# EPICS autosave request: iocBoot/iocCARSPil3Table/auto_settings.req
file "CARS_motor_settings.req",       P=$(P), M=m1
file "CARS_motor_settings.req",       P=$(P), M=m2
file "CARS_motor_settings.req",       P=$(P), M=m3
file "CARS_motor_settings.req",       P=$(P), M=m4
